PROGRAM MAIN
VAR
END_VAR

(* Wanneer de knop wordt ingedrukt, gaat de lamp aan of uit *)
IF GVL_Carbid.Button THEN
   GVL_Carbid.Lamp := TRUE;    (* Zet lamp aan *)
ELSE
    GVL_Carbid.Lamp := FALSE;   (* Zet lamp uit *)
END_IF

END_PROGRAM

(* stored: Version 1.1.0.1, ProductVersion 3.1.4024.12
   POU MAIN: Id {5629203d-57fb-4223-8db4-dc965ae85829}, SpecialFunc None *)
